TYPE ST_HMIKistlerResult :
STRUCT
    eResult     : E_HMIKistlerResult;
    rForce      : REAL;
    rDistance   : REAL;
END_STRUCT
END_TYPE

(* stored: Version 1.1.0.1
   DUT ST_HMIKistlerResult: Id {7f0fb4f6-b57f-42d7-9118-25971f45da18} *)
